FUNCTION "FC_GetNrOfArrayEl" : Int
TITLE = FC_GetNrOfArrayEl
{ S7_Optimized_Access := 'TRUE' }
AUTHOR : MHSE
FAMILY : GeneralSystemFunctions
VERSION : 3.0
// ATTRIBUTES
// AUTO_NUMBER = True
// BLOCK_NUMBER = 19
// END_ATTRIBUTES
//Function to get the number of array elements.
   VAR_INPUT
      iv_Array : Variant;   // Input array
   END_VAR

   VAR_TEMP
      ti_NrOfArrayEl : Int;   // Number of array elements
   END_VAR


BEGIN
	(*
	----------------------------------------------------------------------------------------

	Version history:
	Date        | Version   | Author        | Remark
	----------------------------------------------------------------------------------------
	24/05/2019  | 0.1       | L.Klar        | first release MHS TIA 15.1
	24/07/2019  | 2.0       | L.Klar        | 2.0 MHS library release TIA 15.1
	27/08/2019  | 2.1       | K.Pokorski    | Comments adjusted
	12/11/2019  | 3.0       | P.Majka       | 3.0 MHS library release TIA 15.1
	21/02/2023  | 4.0       | F.Baten       | 4.0 Release TIA 17.5
	*)

	REGION 1 – Number of an array elements

	    IF IS_ARRAY(#iv_Array)                                                  // Input variable is an array
	    THEN

	        #ti_NrOfArrayEl := UDINT_TO_INT(CountOfElements(#iv_Array));

	        // Reset array length if the input variable isn't an array
	    ELSE

	        #ti_NrOfArrayEl := 0;

	    END_IF;

	END_REGION

	REGION 2 – Return output

	    #FC_GetNrOfArrayEl := #ti_NrOfArrayEl;

	END_REGION

END_FUNCTION

